{attribute 'GeneratedUsingTerminal: EKM1101-0000-0016'}
{attribute addProperty BoxType "EKM1101-0000-0016"}
{attribute addProperty Id "StatusAT %I*Status_F2CE6D917ValueAT %I*REAL4"}
{attribute addProperty CRC "1624595570"}
{attribute addProperty Size "11"}
TYPE MMS_Voltage_Up_In_Inputs_60D55C72 EXTENDS InputBase_8311D824 :
STRUCT
	{attribute addProperty Name "Status"}
	Status AT %I* : Status_F2CE6D91;
	{attribute addProperty Name "Value"}
	Value AT %I* : REAL;
END_STRUCT
END_TYPE

(* stored: Version 1.2.0.0, ProductVersion 3.1.4024.9
   DUT MMS_Voltage_Up_In_Inputs_60D55C72: Id {46a68b0a-1d23-4bda-940f-a043b896725f} *)
